Staubli VAL3: SplitMoveJ.pgx

public program SplitMoveJ(string x_sSLine, joint& x_jJ, trsf& x_trP, bool x_bCut, bool& x_bRes)
  local string l_sChar[2]
  local num l_nData[25]
begin
  x_bRes=false

  if x_sSLine==""
    return
  endIf

  x_sSLine=right(x_sSLine,len(x_sSLine)-len("MOVEJ="))

  //解析每一行
  l_sChar[0]=","
  l_sChar[1]="/"

  call SplitNumS(x_sSLine,l_nData,l_sChar,x_bRes)

  if !x_bRes
    return
  endIf

  x_jJ.j1=l_nData[0]
  x_jJ.j2=l_nData[1]
  x_jJ.j3=l_nData[2]
  x_jJ.j4=l_nData[3]
  x_jJ.j5=l_nData[4]
  x_jJ.j6=l_nData[5]



  if !x_bCut

    x_trP.z=l_nData[6]
    x_trP.rx=l_nData[7]
  else
    x_trP.x=l_nData[6]
    x_trP.y=l_nData[7]
    x_trP.z=l_nData[8]
    x_trP.rx=l_nData[9]
    x_trP.ry=l_nData[10]
    //x_trP.rz=l_nData[17]

  endIf




end
